FUNCTION_BLOCK CheckOneBlReady (* Basic Function Block Type *)
  (* Standard: 61499-2 *)
  (* Version 0.0, 7/15/2026, Schneider Electric, Template *)
  PACKAGE SE.Nereda;
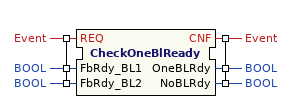
  EVENT_INPUT
    REQ WITH FbRdy_BL1, FbRdy_BL2; (* Normal Execution Request *)
  END_EVENT
  EVENT_OUTPUT
    CNF WITH OneBLRdy, NoBLRdy; (* Execution Confirmation *)
  END_EVENT
  VAR_INPUT
    FbRdy_BL1 : BOOL;
    FbRdy_BL2 : BOOL;
  END_VAR
  VAR_OUTPUT
    OneBLRdy : BOOL;
    NoBLRdy : BOOL;
  END_VAR
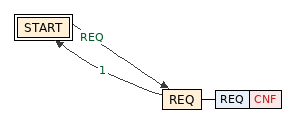
  EC_STATES
    START; (* Initial State *)
    REQ : REQ -> CNF;
  END_STATES
  EC_TRANSITIONS
    START TO REQ := REQ;
    REQ TO START := 1;
  END_TRANSITIONS
  ALGORITHM REQ IN ST: (* Normally executed algorithm *)
;
OneBLRdy := (FbRdy_BL1 AND NOT FbRdy_BL2) OR (NOT FbRdy_BL1 AND FbRdy_BL2);
NoBLRdy := NOT FbRdy_BL1 AND NOT FbRdy_BL2;
  END_ALGORITHM
END_FUNCTION_BLOCK
